KUKA KRL program: turnoffrsi.src, TurnOffRSI.dat

--- turnoffrsi.src ---
&ACCESS RV1
DEF TurnOffRSI (contID:IN)
   INT contID
   INT ret
   RSI_ACTIVE=FALSE
   ret = RSI_OFF()
   IF varstate("contID")==#initialized THEN
      ret = RSI_DELETE(contID)
   ENDIF

END

--- TurnOffRSI.dat ---
&ACCESS RV1
DEFDAT  TurnOffRSI PUBLIC

ENDDAT
